// TwinCAT 3 PLC project nepionic_io
// Title: nepionic-io
// Company: nepionic
// Author: nepionic dev
// ProjectVersion: 0.1.0
// ProgramVersion: 3.1.4024.0
// project tree:
//   Basic/ BasicDigitalOutput.TcPOU, BasicDigitalInput.TcPOU
//   Functions/ AnalogScaler.TcPOU
//   Interfaces/ I_AnalogInput.TcIO, I_DigitalInput.TcIO, I_DigitalOutput.TcIO, I_Overloadable.TcIO, I_Trippable.TcIO, I_TripResettable.TcIO

// ---- Interfaces/I_AnalogInput.TcIO
INTERFACE PUBLIC I_AnalogInput EXTENDS __System.IQueryInterface

{attribute 'monitoring' := 'call'}
PROPERTY PUBLIC Error : BOOL
GET
END_GET
END_PROPERTY

{attribute 'monitoring' := 'call'}
PROPERTY PUBLIC Overrange : BOOL
GET
END_GET
END_PROPERTY

{attribute 'monitoring' := 'call'}
PROPERTY PUBLIC Underrange : BOOL
GET
END_GET
END_PROPERTY

{attribute 'monitoring' := 'call'}
PROPERTY PUBLIC Value : LREAL
GET
END_GET
END_PROPERTY

END_INTERFACE

// ---- Interfaces/I_DigitalInput.TcIO
INTERFACE PUBLIC I_DigitalInput EXTENDS __System.IQueryInterface

{attribute 'monitoring' := 'call'}
PROPERTY PUBLIC State : BOOL
GET
END_GET
END_PROPERTY

END_INTERFACE

// ---- Interfaces/I_DigitalOutput.TcIO
INTERFACE PUBLIC I_DigitalOutput EXTENDS __System.IQueryInterface

{attribute 'monitoring' := 'call'}
PROPERTY PUBLIC State : BOOL
GET
END_GET
SET
END_SET
END_PROPERTY

END_INTERFACE

// ---- Interfaces/I_Overloadable.TcIO
INTERFACE PUBLIC I_Overloadable EXTENDS __System.IQueryInterface

{attribute 'monitoring' := 'call'}
PROPERTY PUBLIC IsOverloaded : BOOL
GET
END_GET
END_PROPERTY

END_INTERFACE

// ---- Interfaces/I_Trippable.TcIO
INTERFACE PUBLIC I_Trippable EXTENDS __System.IQueryInterface

{attribute 'monitoring' := 'call'}
PROPERTY PUBLIC IsTripped : BOOL
GET
END_GET
END_PROPERTY

END_INTERFACE

// ---- Interfaces/I_TripResettable.TcIO
INTERFACE PUBLIC I_TripResettable EXTENDS __System.IQueryInterface

METHOD TripReset : BOOL
END_METHOD

END_INTERFACE

// ---- Basic/BasicDigitalOutput.TcPOU
{attribute 'linkalways'} 
{attribute 'no_explicit_call' := 'This FB is a CLASS and must be accessed using methods or properties'}
{attribute 'enable_dynamic_creation'}
FUNCTION_BLOCK PUBLIC BasicDigitalOutput IMPLEMENTS I_DigitalOutput
VAR
	output AT %Q* : BOOL;
	inverted : BOOL;
END_VAR

METHOD FB_init : BOOL
VAR_INPUT
	bInitRetains : BOOL; // if TRUE, the retain variables are initialized (warm start / cold start)
	bInCopyCode : BOOL;  // if TRUE, the instance afterwards gets moved into the copy code (online change)
	inverted : BOOL;
END_VAR
THIS^.inverted := inverted;
END_METHOD

{attribute 'monitoring' := 'call'}
PROPERTY PUBLIC State : BOOL
GET // PUBLIC
State := output XOR inverted;
END_GET
SET // PUBLIC
output := State XOR inverted;
END_SET
END_PROPERTY

END_FUNCTION_BLOCK

// ---- Basic/BasicDigitalInput.TcPOU
{attribute 'linkalways'} 
{attribute 'no_explicit_call' := 'This FB is a CLASS and must be accessed using methods or properties'}
{attribute 'enable_dynamic_creation'}
FUNCTION_BLOCK PUBLIC BasicDigitalInput IMPLEMENTS I_DigitalInput
VAR
	input AT %Q* : BOOL;
	inverted : BOOL;
END_VAR

METHOD FB_init : BOOL
VAR_INPUT
	bInitRetains : BOOL; // if TRUE, the retain variables are initialized (warm start / cold start)
	bInCopyCode : BOOL;  // if TRUE, the instance afterwards gets moved into the copy code (online change)
	inverted : BOOL;
END_VAR
THIS^.inverted := inverted;
END_METHOD

{attribute 'monitoring' := 'call'}
PROPERTY PUBLIC State : BOOL
GET // PUBLIC
State := input XOR inverted;
END_GET
END_PROPERTY

END_FUNCTION_BLOCK

// ---- Functions/AnalogScaler.TcPOU
FUNCTION AnalogScaler : LREAL
VAR_INPUT
	input : LREAL;
	rawLow : LREAL;
	rawHigh : LREAL;
	processLow : LREAL;
	processHigh : LREAL;
END_VAR

AnalogScaler := (processHigh - processLow)
	* (input - rawLow)
	/ (rawHigh - rawLow)
	+ processLow;

END_FUNCTION
